(* PLC project Unnamed, Unknown Unnamed 1 *)
(* stored: creationDateTime 2020-05-29T13:29:11, modificationDateTime 2020-06-02T18:39:50 *)

PROGRAM RPi
  VAR
    presure_sensor AT %IW100 : UINT;
    temp_sensor AT %IW101 : UINT;
    relay AT %QX100.0 : BOOL;
  END_VAR

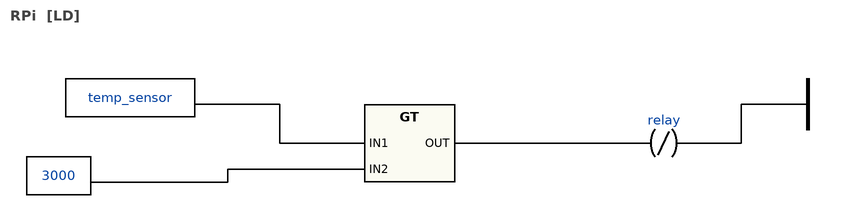
(* LD diagram, written out as Structured Text *)
relay := NOT (temp_sensor > 3000);
END_PROGRAM

CONFIGURATION Config0
  RESOURCE Res0 ON PLC
    TASK task0(INTERVAL := T#20ms, PRIORITY := 0);
    PROGRAM instance0 WITH task0 : RPi;
  END_RESOURCE
END_CONFIGURATION
